// TwinCAT 3 PLC project PID
// ProgramVersion: 3.1.4023.0
// libraries:
//   Tc2_Standard, * (Beckhoff Automation GmbH)
//   Tc2_System, * (Beckhoff Automation GmbH)
//   Tc3_Module, * (Beckhoff Automation GmbH)
// project tree:
//   / PlcTask.TcTTO
//   POUs/ MAIN.TcPOU
//   POUs/PID/ FB_PID.TcPOU, GVL_PID.TcGVL, rt_floord.TcPOU
// real-time tasks:
//   TASK PlcTask: cycle T#10ms, priority 20, ADS port 350

CONFIGURATION PID
    RESOURCE PLC ON TwinCAT3
        TASK PlcTask(INTERVAL := T#10ms, PRIORITY := 20);
        PROGRAM MAIN WITH PlcTask : MAIN;
    END_RESOURCE
END_CONFIGURATION

// ---- POUs/PID/GVL_PID.TcGVL
VAR_GLOBAL CONSTANT
	nInitialize: SINT := 0;
	nStep: SINT := 1;
END_VAR

// ---- POUs/MAIN.TcPOU
PROGRAM MAIN
VAR
	//Inputs
	fb_PIDController :	FB_PID;			
	fIn	: LREAL;				
	fKp	: LREAL := 0.5;				
	fKi	: LREAL := 0.1;				
	fKd	: LREAL := 0.01;				
	fSatHigh : LREAL := 100.0;		
	fSatLow	 : LREAL := -100.0;		
	bReset: BOOL;	
	
	//Output 
	fPIDOut	: LREAL;	
END_VAR

fb_PIDController(nMethodType:= GVL_PID.nStep,
				 fIn := fIn,
				 fKp := fKp,
				 fKi := fKi,
				 fKd := fKd,
				 fSatHigh := fSatHigh,
				 fSatLow := fSatLow,
				 bReset := bReset,
				 fPIDOutput => fPIDOut);

END_PROGRAM

// ---- POUs/PID/FB_PID.TcPOU
FUNCTION_BLOCK FB_PID
VAR_INPUT
	nMethodType: SINT;		//Method tpye: '0' for initialization, '1' for start-up
	fIn: LREAL;				//Controller input 
	fKp: LREAL;				//Proportional gain
	fKi: LREAL;				//Integral gain
	fKd: LREAL;				//Derivative gain
	fSatHigh : LREAL;		//High saturation limit
	fSatLow	 : LREAL;		//Low saturation limit	
	bReset: BOOL;			//PID internal reset
END_VAR
VAR_OUTPUT
	fPidOutput: LREAL;	
END_VAR
VAR
	rtb_Sum: LREAL;
	rtb_TSamp: LREAL;
	UD_DSTATE: LREAL;
	Integrator_PrevResetState: SINT;
	Integrator_DState: LREAL;
	UD_Reset_ZCE: USINT := 1;
END_VAR

CASE nMethodType OF
    nInitialize: 
       //Initialize conditions for discrete integrator
        Integrator_DState := 0.0;
        Integrator_PrevResetState := 2;
        //InitializeConditions for delay
        UD_DSTATE := 0.0;
    nStep: 
        //Discrete integrator
        IF bReset AND (Integrator_PrevResetState <= 0) THEN 
            Integrator_DState := 0.0;
        END_IF;
        
        // y = u * K where K = 1 / ( w * Ts ) *)
        rtb_TSamp := (fIn * fKd) * 20.0;  

        IF bReset AND (UD_Reset_ZCE <> 1) THEN 
            UD_DSTATE := 0.0;
        END_IF;

        UD_Reset_ZCE := BOOL_TO_USINT(bReset);
        
        rtb_Sum := ((fIn * fKp) + Integrator_DState) + (rtb_TSamp - UD_DSTATE);		
        
		// Saturation limits
        IF rtb_Sum >= fSatHigh THEN 
            fPidOutput := fSatHigh;
        ELSIF rtb_Sum > fSatLow THEN 
            fPidOutput := rtb_Sum;
        ELSE 
            fPidOutput := 0.0;
        END_IF;       

        // Update for discrete integrator        
        Integrator_DState := (((fIn * fKi) + (fPidOutput - rtb_Sum)) * 0.05) + Integrator_DState;

        IF bReset THEN 
            Integrator_PrevResetState := 1;
        ELSE 
            Integrator_PrevResetState := 0;
        END_IF;       

        //Update for delay
        UD_DSTATE := rtb_TSamp;
END_CASE;

END_FUNCTION_BLOCK

// ---- POUs/PID/rt_floord.TcPOU
FUNCTION rt_floord : LREAL
VAR_INPUT
	u: LREAL;
END_VAR
VAR
END_VAR

rt_floord := DINT_TO_LREAL(TRUNC(u));
IF u = rt_floord THEN 
    rt_floord := u;
ELSIF u < 0.0 THEN 
    rt_floord := rt_floord - 1.0;
END_IF;

END_FUNCTION
